INTERFACE ITF_BaseLoggerElement_HMI_Connector_Command

END_INTERFACE

(* stored: Version 1.1.0.1
   Itf ITF_BaseLoggerElement_HMI_Connector_Command: Id {26cd0ad0-561e-081a-2614-e63e2addf549} *)
